TYPE TYP_HW_L4000_IN :
STRUCT
	AcqStatus : TYP_HW_L4000_ACQ_STATUS;
	InspStatus : TYP_HW_L4000_INSP_STATUS;
	CommandResult AT %I* : UINT;
	ExternalEvent : TYP_HW_L4000_EXT_STATUS;
	InspResults : TYP_HW_L4000_INSP_RESULTS;
END_STRUCT
END_TYPE

(* stored: Version 1.1.0.1, ProductVersion 3.1.4024.12
   DUT TYP_HW_L4000_IN: Id {0cca398b-f79f-49b4-9636-e50542517715} *)
